// TIA Portal V18 export
TYPE "LGasp_typeTrackingPart"
// stored: IsFailsafeCompliant false
   STRUCT
      num_pezzo : DInt;   // Numero pezzo
      tipologia : DInt;   // Tipo di profilo
      nome_articolo : String["NumCharTrackingArticle"];   // nome articolo
      lotto : String["NumCharTrackingLotto"];   // nome lotto
      ID_riga : DInt;   // Compone il pacco
      lunghezza : LReal;   // lunghezza [mm]
      larghezza : LReal;   // larghezza [mm]
      altezza : LReal;   // altezza [mm]
      spessore : LReal;   // spessore [mm]
      testo_stampa : WString;   // testo da stampare
      layout_stampa : WString;   // layout da impostare
      qualita_pezzo : Int;   // qualità del pezzo (buono, seconda scelta, scarto)
      options : Array[1..16] of Bool;   // dati aggiuntivi pezzo tracking
      options_str : Array[1..3] of WString[20];   // dati aggiuntivi pezzo tracking
      options_lreal : Array[1..3] of LReal;   // dati aggiuntivi pezzo tracking
      options_dint : Array[1..3] of DInt;   // dati aggiuntivi pezzo tracking
   END_STRUCT;
END_TYPE
